(* CODESYS project mobject-basic-nodepack.library
   Company: mobject
   DefaultNamespace: mobject-basic-nodepack
   Version: 0.2.0
   Placeholder: mobject-basic-nodepack
   Author: mobject dev team
   Title: mobject-basic-nodepack

Project tree, tasks and I/O mapping:
  libraries: mobject-basic-datatypes, 0.2.0 (mobject); mobject-graph, 0.2.0 (mobject); mobject-datatypes, 0.5.0 (mobject)
  Display/
    function block BooleanDisplayNode [ST]: FB_init, Clone, OnExecute
    function block IntDisplayNode [ST]: FB_init, Clone, OnExecute
    function block RealDisplayNode [ST]: FB_init, Clone, OnExecute
  Hardware/
    function block DigitalInputNode [ST]: FB_init, Clone, Dispose, OnExecute
    function block DigitalOutputNode [ST]: FB_init, Clone, Dispose, OnExecute
  Literals/
    function block BooleanLiteralNode [ST]: FB_init, Clone, OnExecute
    function block IntLiteralNode [ST]: FB_init, Clone, OnExecute
    function block RealLiteralNode [ST]: FB_init, Clone, OnExecute
  function block BasicNodePack [ST]: RegisterWithNodeFactory
*)

// Display/BooleanDisplayNode
{attribute 'linkalways'} 
{attribute 'no_explicit_call' := 'This FB is a CLASS and must be accessed using methods or properties'}
{attribute 'enable_dynamic_creation'}
FUNCTION_BLOCK FINAL BooleanDisplayNode EXTENDS Node
VAR
	in : _BOOL(FALSE);
	display : _BOOL(FALSE);
END_VAR

METHOD FB_init : BOOL
VAR_INPUT
	bInitRetains : BOOL; // if TRUE, the retain variables are initialized (warm start / cold start)
	bInCopyCode : BOOL;  // if TRUE, the instance afterwards gets moved into the copy code (online change)
END_VAR
AddInput('in', in);
AddContent('display', display);
END_METHOD

METHOD PUBLIC Clone : I_Node
VAR
	pNode : POINTER TO BooleanDisplayNode;
END_VAR
pNode := __NEW(BooleanDisplayNode);
Clone := pNode^;
END_METHOD

METHOD PROTECTED OnExecute : HRESULT
display.Value := in.Value;
END_METHOD

END_FUNCTION_BLOCK

// Display/IntDisplayNode
{attribute 'linkalways'} 
{attribute 'no_explicit_call' := 'This FB is a CLASS and must be accessed using methods or properties'}
{attribute 'enable_dynamic_creation'}
FUNCTION_BLOCK FINAL IntDisplayNode EXTENDS Node
VAR
	in : _INT(0);
	display : _INT(0);
END_VAR

METHOD FB_init : BOOL
VAR_INPUT
	bInitRetains : BOOL; // if TRUE, the retain variables are initialized (warm start / cold start)
	bInCopyCode : BOOL;  // if TRUE, the instance afterwards gets moved into the copy code (online change)
END_VAR
AddInput('in', in);
AddContent('display', display);
END_METHOD

METHOD PUBLIC Clone : I_Node
VAR
	pNode : POINTER TO IntDisplayNode;
END_VAR
pNode := __NEW(IntDisplayNode);
Clone := pNode^;
END_METHOD

METHOD PROTECTED OnExecute : HRESULT
display.Value := in.Value;
END_METHOD

END_FUNCTION_BLOCK

// Display/RealDisplayNode
{attribute 'linkalways'} 
{attribute 'no_explicit_call' := 'This FB is a CLASS and must be accessed using methods or properties'}
{attribute 'enable_dynamic_creation'}
FUNCTION_BLOCK FINAL RealDisplayNode EXTENDS Node
VAR
	in : _REAL(0.0);
	display : _REAL(0.0);
END_VAR

METHOD FB_init : BOOL
VAR_INPUT
	bInitRetains : BOOL; // if TRUE, the retain variables are initialized (warm start / cold start)
	bInCopyCode : BOOL;  // if TRUE, the instance afterwards gets moved into the copy code (online change)
END_VAR
AddInput('in', in);
AddContent('display', display);
END_METHOD

METHOD PUBLIC Clone : I_Node
VAR
	pNode : POINTER TO RealDisplayNode;
END_VAR
pNode := __NEW(RealDisplayNode);
Clone := pNode^;
END_METHOD

METHOD PROTECTED OnExecute : HRESULT
display.Value := in.Value;
END_METHOD

END_FUNCTION_BLOCK

// Hardware/DigitalInputNode
{attribute 'linkalways'} 
{attribute 'no_explicit_call' := 'This FB is a CLASS and must be accessed using methods or properties'}
{attribute 'enable_dynamic_creation'}
FUNCTION_BLOCK FINAL DigitalInputNode EXTENDS Node
VAR
	input AT %I* : BOOL;
	out : _BOOL(FALSE);
END_VAR

METHOD FB_init : BOOL
VAR_INPUT
	bInitRetains : BOOL; // if TRUE, the retain variables are initialized (warm start / cold start)
	bInCopyCode : BOOL;  // if TRUE, the instance afterwards gets moved into the copy code (online change)
END_VAR
AddOutput('out', out);
END_METHOD

METHOD PUBLIC Clone : I_Node
VAR
END_VAR
Clone := this^;
END_METHOD

METHOD Dispose
VAR_INPUT
END_VAR
END_METHOD

METHOD PROTECTED OnExecute : HRESULT
VAR
END_VAR
out.value := input;
END_METHOD

END_FUNCTION_BLOCK

// Hardware/DigitalOutputNode
{attribute 'linkalways'} 
{attribute 'no_explicit_call' := 'This FB is a CLASS and must be accessed using methods or properties'}
{attribute 'enable_dynamic_creation'}
FUNCTION_BLOCK FINAL DigitalOutputNode EXTENDS Node
VAR
	output AT %Q* : BOOL;
	in : _BOOL(FALSE);
END_VAR

METHOD FB_init : BOOL
VAR_INPUT
	bInitRetains : BOOL; // if TRUE, the retain variables are initialized (warm start / cold start)
	bInCopyCode : BOOL;  // if TRUE, the instance afterwards gets moved into the copy code (online change)
END_VAR
AddInput('in', in);
END_METHOD

METHOD PUBLIC Clone : I_Node
VAR
END_VAR
Clone := this^;
END_METHOD

METHOD Dispose
VAR_INPUT
END_VAR
END_METHOD

METHOD PROTECTED OnExecute : HRESULT
VAR
END_VAR
output := in.value;
END_METHOD

END_FUNCTION_BLOCK

// Literals/BooleanLiteralNode
{attribute 'linkalways'} 
{attribute 'no_explicit_call' := 'This FB is a CLASS and must be accessed using methods or properties'}
{attribute 'enable_dynamic_creation'}
FUNCTION_BLOCK FINAL BooleanLiteralNode EXTENDS Node
VAR
	value : _BOOL(FALSE);
	out : _BOOL(FALSE);
END_VAR

METHOD FB_init : BOOL
VAR_INPUT
	bInitRetains : BOOL; // if TRUE, the retain variables are initialized (warm start / cold start)
	bInCopyCode : BOOL;  // if TRUE, the instance afterwards gets moved into the copy code (online change)
END_VAR
AddParameter('value', value);
AddOutput('out', out);
END_METHOD

METHOD PUBLIC Clone : I_Node
VAR
	pNode : POINTER TO BooleanLiteralNode;
END_VAR
pNode := __NEW(BooleanLiteralNode);
Clone := pNode^;
END_METHOD

METHOD PROTECTED OnExecute : HRESULT
VAR
END_VAR
out.value := value.value;
END_METHOD

END_FUNCTION_BLOCK

// Literals/IntLiteralNode
{attribute 'linkalways'} 
{attribute 'no_explicit_call' := 'This FB is a CLASS and must be accessed using methods or properties'}
{attribute 'enable_dynamic_creation'}
FUNCTION_BLOCK FINAL IntLiteralNode EXTENDS Node
VAR
	value : _INT(0);
	out : _INT(0);
END_VAR

METHOD FB_init : BOOL
VAR_INPUT
	bInitRetains : BOOL; // if TRUE, the retain variables are initialized (warm start / cold start)
	bInCopyCode : BOOL;  // if TRUE, the instance afterwards gets moved into the copy code (online change)
END_VAR
AddParameter('value', value);
AddOutput('out', out);
END_METHOD

METHOD PUBLIC Clone : I_Node
VAR
	pNode : POINTER TO IntLiteralNode;
END_VAR
pNode := __NEW(IntLiteralNode);
Clone := pNode^;
END_METHOD

METHOD PROTECTED OnExecute : HRESULT
VAR
END_VAR
out.value := value.value;
END_METHOD

END_FUNCTION_BLOCK

// Literals/RealLiteralNode
{attribute 'linkalways'} 
{attribute 'no_explicit_call' := 'This FB is a CLASS and must be accessed using methods or properties'}
{attribute 'enable_dynamic_creation'}
FUNCTION_BLOCK FINAL RealLiteralNode EXTENDS Node
VAR
	value : _REAL(0.0);
	out : _REAL(0.0);
END_VAR

METHOD FB_init : BOOL
VAR_INPUT
	bInitRetains : BOOL; // if TRUE, the retain variables are initialized (warm start / cold start)
	bInCopyCode : BOOL;  // if TRUE, the instance afterwards gets moved into the copy code (online change)
END_VAR
AddParameter('value', value);
AddOutput('out', out);
END_METHOD

METHOD PUBLIC Clone : I_Node
VAR
	pNode : POINTER TO RealLiteralNode;
END_VAR
pNode := __NEW(RealLiteralNode);
Clone := pNode^;
END_METHOD

METHOD PROTECTED OnExecute : HRESULT
VAR
END_VAR
out.value := value.value;
END_METHOD

END_FUNCTION_BLOCK

// BasicNodePack
{attribute 'linkalways'} 
{attribute 'no_explicit_call' := 'This FB is a CLASS and must be accessed using methods or properties'}
{attribute 'enable_dynamic_creation'}
FUNCTION_BLOCK BasicNodePack IMPLEMENTS I_NodePack
VAR
	booleanLiteralNode : BooleanLiteralNode;
	booleanDisplayNode : BooleanDisplayNode;
	intLiteralNode : IntLiteralNode;
	intDisplayNode : IntDisplayNode;
	realLiteralNode : RealLiteralNode;
	realDisplayNode : RealDisplayNode;
END_VAR

METHOD PUBLIC RegisterWithNodeFactory
VAR_INPUT
	NodeFactory : I_NodeFactory;
END_VAR
NodeFactory.AddNodeAsPrototype('PlcBasic.Bool.BoolLiteral',booleanLiteralNode);
NodeFactory.AddNodeAsPrototype('PlcBasic.Bool.BoolDisplay',booleanDisplayNode);
NodeFactory.AddNodeAsPrototype('PlcBasic.Int.IntLiteral',intLiteralNode);
NodeFactory.AddNodeAsPrototype('PlcBasic.Int.IntDisplay',intDisplayNode);
NodeFactory.AddNodeAsPrototype('PlcBasic.Real.RealLiteral',realLiteralNode);
NodeFactory.AddNodeAsPrototype('PlcBasic.Real.RealDisplay',realDisplayNode);
END_METHOD

END_FUNCTION_BLOCK
